// TwinCAT 3 PLC project Untitled1
// ProgramVersion: 3.1.4020.2
// libraries:
//   Tc2_Standard, * (Beckhoff Automation GmbH)
//   Tc2_System, * (Beckhoff Automation GmbH)
//   Tc3_Module, * (Beckhoff Automation GmbH)
// project tree:
//   DUTs/ ST_Record.TcDUT
//   GVLs/ GVL.TcGVL
//   / PlcTask.TcTTO
//   POUs/ FB_AdsSend.TcPOU, MAIN.TcPOU
// real-time tasks:
//   TASK PlcTask: cycle T#10ms, priority 20, ADS port 350

CONFIGURATION Untitled1
    RESOURCE PLC ON TwinCAT3
        TASK PlcTask(INTERVAL := T#10ms, PRIORITY := 20);
        PROGRAM MAIN WITH PlcTask : MAIN;
    END_RESOURCE
END_CONFIGURATION

// ---- DUTs/ST_Record.TcDUT
TYPE ST_Record :
STRUCT
	test : ARRAY[0..99999] OF DWORD;
	test2 : ARRAY[0..99999] OF DWORD;
	test3 : ARRAY[0..99999] OF DWORD;
END_STRUCT
END_TYPE

// ---- GVLs/GVL.TcGVL
{attribute 'qualified_only'}
VAR_GLOBAL
	NetId: STRING := '5.31.27.244.1.1';
	Port : UINT := 851;
	Timeout : TIME := T#5S;
END_VAR

// ---- POUs/MAIN.TcPOU
PROGRAM MAIN
VAR
	record : ST_Record;
	counter : INT;
	
	adsSendData : FB_AdsSend;
	
	start: BOOL;
	random: BOOL;
	randomize : DRAND;
	
	i: INT;
	timer : TON := (IN := TRUE);
	bBusy: BOOL;
	nState: INT;
END_VAR

(*-------- Put dummy value to be sent --------*)
IF random THEN
	FOR i := 0 TO 10000 DO
		randomize(Seed:= 0 , Num=> );
		record.test[i] := LREAL_TO_DWORD(randomize.Num * 100);
		record.test2[i] := LREAL_TO_DWORD(randomize.Num * 100);
		record.test3[i] := LREAL_TO_DWORD(randomize.Num * 100);
	END_FOR
END_IF


(*-------- Send data every second --------*)
timer(IN:= , PT:= T#1000MS, Q=> , ET=> );
IF timer.Q THEN
	nState := 0;
	timer.IN := FALSE;
END_IF


adsSendData(SendVarLen := SIZEOF(record), SendVarAddr:= ADR(record), TargetVarName:= 'MAIN.record');

CASE nState OF 
	0:
	adsSendData.bStart := TRUE;
	nState := 10;
	
	10:
	IF NOT adsSendData.bBusy OR adsSendData.bError THEN
		adsSendData.bStart := FALSE;
		timer.IN := TRUE;
	END_IF
END_CASE

END_PROGRAM

// ---- POUs/FB_AdsSend.TcPOU
FUNCTION_BLOCK FB_AdsSend
VAR_INPUT
	
	SendVarLen: UDINT;
	SendVarAddr: POINTER TO ST_Record;
	TargetVarName: STRING;
	bStart : BOOL;
END_VAR
VAR_OUTPUT
	bBusy : BOOL;
	bError: BOOL;
	nErrId: UDINT;
END_VAR
VAR
	adsRdWrt : ADSRDWRT;
	adsWrt1 : ADSWRITE;
	adsWrt2 : ADSWRITE;
	
	iSendVar : ARRAY[0..9999] OF DWORD;
	nameVar : STRING := 'MAIN.test';
	handleVar : UDINT;
	
	ADSRDWRT1RDWRT: BOOL;
	Write: BOOL;
	WriteDeleteHandle: BOOL;
	
	state : INT;
	
	trig : R_TRIG;
	counter: INT;
END_VAR

trig(CLK := bStart);

//create handle
adsRdWrt(
	NETID:= GVL.NetId, 
	PORT:= GVL.Port, 
	IDXGRP:= 16#F003, 
	IDXOFFS:= 0, 
	WRITELEN:= LEN(TargetVarName)+1, 
	READLEN:= SIZEOF(handleVar), 
	SRCADDR:= ADR(TargetVarName), 
	DESTADDR:= ADR(handleVar), 
	WRTRD:= , 
	TMOUT:= GVL.Timeout, 
	BUSY=> bBusy, 
	ERR=> bError, 
	ERRID=> nErrId);

//write to handle
adsWrt1(
	NETID:= GVL.NetId, 
	PORT:= GVL.Port, 
	IDXGRP:= 16#F005, 
	IDXOFFS:= handleVar, 
	LEN:= SendVarLen, 
	SRCADDR:= SendVarAddr, 
	WRITE:= , 
	TMOUT:= GVL.Timeout, 
	BUSY=> bBusy, 
	ERR=> bError, 
	ERRID=> nErrId);
	
//delete handle
adsWrt2(
	NETID:= GVL.NetId, 
	PORT:= GVL.Port, 
	IDXGRP:= 16#F006, 
	IDXOFFS:= 0, 
	LEN:= SIZEOF(handleVar), 
	SRCADDR:= ADR(handleVar), 
	WRITE:= , 
	TMOUT:= GVL.Timeout, 
	BUSY=> bBusy, 
	ERR=> bError, 
	ERRID=> nErrId);
			
IF trig.q THEN
	state := 0;
END_IF

CASE state OF 
	//create handle
	0:
	adsRdWrt.WRTRD := TRUE;
	state := 10;
	
	10:
	IF NOT adsRdWrt.BUSY OR adsRdWrt.ERR THEN
		adsRdWrt.WRTRD := FALSE;
		state := 20;
	END_IF	
	
	//Write to handle
	20:
	adsWrt1.WRITE := TRUE;
	state := 30;
	
	30:
	IF NOT adsWrt1.BUSY OR adsWrt1.ERR THEN
		adsWrt1.WRITE := FALSE;
		state := 40;
	END_IF
	
	//Delete handle
	40:
	adsWrt2.WRITE := TRUE;
	state := 50;
	
	50:
	IF NOT adsWrt2.BUSY OR adsWrt2.ERR THEN
		adsWrt2.WRITE := FALSE;
		state := 60;
	END_IF
	
END_CASE

END_FUNCTION_BLOCK
